{attribute addProperty BoxType "ELM9410-0000-0016"}
{attribute addProperty Id "StatusAT %I*Status_050B615A81"}
{attribute addProperty CRC "2215490587"}
{attribute addProperty SizeInBites "8"}
{attribute addProperty SizeInBytes "1"}
TYPE MMS_Device_Inputs_840DB41B :
STRUCT
	{attribute addProperty Name "Status"}
	Status AT %I* : Status_050B615A;
END_STRUCT
END_TYPE

(* stored: Version 1.2.0.0, ProductVersion 3.1.4024.9
   DUT MMS_Device_Inputs_840DB41B: Id {3ef538a3-f5fc-4ba6-b311-3fc081f3865e} *)
